(*
Casts I_Component as I_Tagged.
Returns:
- Ok - Success,
- Err.InvRef - Invalid reference,
- Err.Itf0 - Invalid interface,
- Err.NoMatch - Cast failed
*)
FUNCTION ICompToITagged : Result
VAR_INPUT
	iIn		: I_RawComponent;
	iOut	: REFERENCE TO I_Tagged;
END_VAR

IF NOT __ISVALIDREF(iOut) THEN
	ICompToITagged := Err.InvRef;
	RETURN;
END_IF

IF iIn = 0 THEN
	ICompToITagged := Err.Itf0;
	RETURN;
END_IF

IF __QUERYINTERFACE(iIn, iOut) THEN
	ICompToITagged := Ok;
ELSE
	ICompToITagged := Err.NoMatch;
END_IF

END_FUNCTION

(* stored: Version 1.1.0.1
   POU ICompToITagged: Id {037a1bf0-02fe-469d-a7f0-fdd83b19b2c8}, SpecialFunc None *)
